PROGRAM main
  VAR
    tank_level : INT := 50;
    pump_on : BOOL := FALSE;
    low_level : BOOL := FALSE;
    high_level : BOOL := FALSE;
    RS0 : RS;
  END_VAR

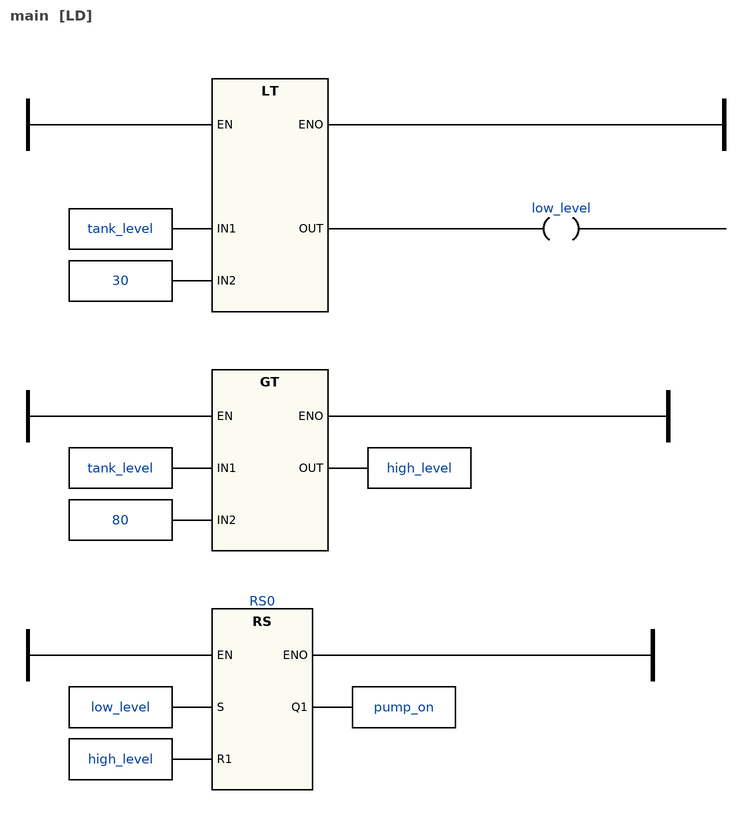
(* LD diagram, written out as Structured Text *)
low_level := tank_level < 30;
high_level := tank_level > 80;
RS0(S := low_level, R1 := high_level);
pump_on := RS0.Q1;
END_PROGRAM
